FUNCTION_BLOCK T_ModuleCollectionNotifyStateChangedSuccess EXTENDS T_UnitTestBase
VAR
  list : T_SubModuleCollection(10);
  newModule, newModule2 : T_SubModuleMock; 
  actual1, actual2 : BOOL;
END_VAR

// Arrange
list.AddModule(newModule);
list.AddModule(newModule2);

//Act
list.NotifyStateChanged(Tc3_PackML_V2.E_PMLCommand.ePMLCommand_Complete);

//Assert
actual1 := newModule._newState = Tc3_PackML_V2.E_PMLCommand.ePMLCommand_Complete;
actual2 := newModule2._newState = Tc3_PackML_V2.E_PMLCommand.ePMLCommand_Complete;

assertion.AssertEquals_BOOL(TRUE, actual1, 'newModule._newState = Tc3_PackML_V2.E_PMLCommand.ePMLCommand_Complete');
assertion.AssertEquals_BOOL(TRUE, actual2, 'newModule._newState = Tc3_PackML_V2.E_PMLCommand.ePMLCommand_Complete');
TestFinished();

END_FUNCTION_BLOCK

(* stored: Version 1.1.0.1, ProductVersion 3.1.4024.12
   POU T_ModuleCollectionNotifyStateChangedSuccess: Id {d29cb869-5caf-4c39-98b9-e59bcec99999}, SpecialFunc None *)
